FUNCTION_BLOCK PUBLIC Trigger
VAR_INPUT
END_VAR
VAR_OUTPUT
END_VAR
VAR
	{attribute 'OPC.UA.DA' := '0'}
	_logger : Logger;
	{attribute 'OPC.UA.DA' := '0'}
	_message : StringBuilder;
	
	{attribute 'OPC.UA.DA' := '0'}
	_execStartTrigger : BOOL;

	{attribute 'OPC.UA.DA' := '0'}
	_stateCmd : INT;
	{attribute 'OPC.UA.DA' := '0'}
	_setPeriod_ms : LREAL;
	
	{attribute 'OPC.UA.DA' := '0'}
	timerDelayOn : TON;
	{attribute 'OPC.UA.DA' := '0'}
	timerDelayOff: TON;	
	{attribute 'OPC.UA.DA' := '0'}
	pulseFlag : BOOL;
	{attribute 'OPC.UA.DA' := '0'}	
	trigOff : BOOL;	
	{attribute 'OPC.UA.DA' := '0'}
	OutputTrigger	AT %Q* : BOOL;	
END_VAR

TriggerOutEmitSignal(_execStartTrigger, _setPeriod_ms);

{attribute 'TcRpcEnable' := '1'}
METHOD PROTECTED TriggerOutEmitSignal
VAR_INPUT
	Execute : BOOL;
	PulseDuration_ms : LREAL;	
END_VAR
VAR
	demiPulseDuration_ms : TIME;
END_VAR
(*
// La FastTask a un cycle de 50µs. Il faut 4 instructions pour obtenir un pulse.
// On aura donc un pulse minimum de 200 µs (4 * 50 µs) 
*)

IF Execute THEN
	_execStartTrigger := TRUE;
	_setPeriod_ms := PulseDuration_ms;
	
	demiPulseDuration_ms := LREAL_TO_TIME(_setPeriod_ms * 1E+6) / 2;
	
	_logger.Information(_message.Reset().Append('TriggerOutEmitSignal').ToString());
	
	CASE _stateCmd OF
		0:  timerDelayOn(IN := _execStartTrigger AND NOT trigOff, PT := demiPulseDuration_ms);
			OutputTrigger := timerDelayOn.Q;
			
			timerDelayOff(IN := OutputTrigger, PT := demiPulseDuration_ms);
			trigOff := timerDelayOff.Q;
				
			//_execStartTrigger := FALSE;
	END_CASE
END_IF
END_METHOD

END_FUNCTION_BLOCK

(* stored: Version 1.1.0.1, ProductVersion 3.1.4024.12
   POU Trigger: Id {586c7298-54a8-43f3-b1e3-5df1e7eac297}, SpecialFunc None
   Method TriggerOutEmitSignal: Id {0402d862-386b-4b9d-a2a1-b19a7ce5488c} *)
